// Mitsubishi GX Works2 project: 26 unfinish   PLC: FX3G

// task Task_01 (event TRUE, interval 0, priority 31): POU_01

PROGRAM POU_01
VAR
  gas : INT;
  ton1 : TON;
END_VAR
IF M8002 THEN
	gas := 0;
END_IF;
IF M0 THEN 
	gas:=0;
Y0:=FALSE;
Y1:=FALSE;
Y2:=FALSE;
Y3:=FALSE;
END_IF;

IF M7 THEN
		gas:=99;
END_IF;


CASE gas OF
0:
IF M1 THEN 
	gas:=1;
	END_IF;

1:
Y0:=TRUE;
IF M2 THEN 
	gas:=2;
END_IF;
IF M3 THEN 
	gas:=10;
END_IF;

2:
IF M6 THEN
	gas:=3;
END_IF;

3:
Y0:=FALSE;
Y3:=TRUE;
ton1(IN := NOT ton1.Q, PT := T#20s);
	IF ton1.Q THEN
		gas:=4;
	END_IF;
	 
4:
Y3:=FALSE;
IF M7 THEN 
	gas:=0;
END_IF;

10:
IF M4 THEN 
	gas:=11;
END_IF;

11:
Y0:=FALSE;
Y1:=TRUE;
ton1(IN := NOT ton1.Q, PT := T#5s);
	IF ton1.Q THEN
		gas:=12;
	END_IF;
	
12:
Y0:=TRUE;
Y1:=FALSE;
IF M5 THEN 
	gas:=13;
END_IF;

13:
Y0:=FALSE;
Y2:=TRUE;
ton1(IN := NOT ton1.Q, PT := T#15s);
	IF ton1.Q THEN
		gas:=14;
	END_IF;

14:
Y0:=TRUE;
Y2:=FALSE;
IF M6 THEN
	gas:=15;
END_IF;

15:
Y0:=FALSE;
Y3:=TRUE;
ton1(IN := NOT ton1.Q, PT := T#20s);
	IF ton1.Q THEN
		gas:=0;
	END_IF;

99:
Y0:=FALSE;
Y1:=FALSE;
Y2:=FALSE;
Y3:=FALSE;
IF NOT M7 THEN
	gas:=0;
	END_IF;
END_CASE;
END_PROGRAM
